// TIA Portal project "Connection" (V15.1)

(* hardware
DEVICE "S71500/ET200MP station_1"  S7-1500 station
   slot 0: "PM 190W 120/230VAC"  PM 190W 120/230VAC  6EP1333-4BA00
   slot 0: "Rail_0"  Rack  6ES7 590-1***0-0AA0
   slot 1: "PLC_1"  CPU 1516-3 PN/DP  6ES7 516-3AN01-0AB0  V2.6
      slot 3: "CPU display_1"  6ES7591-1BA00-0AA0
*)

// ===== PLC "PLC_1"  CPU 1516-3 PN/DP =====

VAR_GLOBAL   // PLC tag table "Default tag table"
   "System_Byte" AT %MB1 : Byte;
   "FirstScan" AT %M1.0 : Bool;
   "DiagStatusUpdate" AT %M1.1 : Bool;
   "AlwaysTRUE" AT %M1.2 : Bool;
   "AlwaysFALSE" AT %M1.3 : Bool;
   "Clock_Byte" AT %MB0 : Byte;
   "Clock_10Hz" AT %M0.0 : Bool;
   "Clock_5Hz" AT %M0.1 : Bool;
   "Clock_2.5Hz" AT %M0.2 : Bool;
   "Clock_2Hz" AT %M0.3 : Bool;
   "Clock_1.25Hz" AT %M0.4 : Bool;
   "Clock_1Hz" AT %M0.5 : Bool;
   "Clock_0.625Hz" AT %M0.6 : Bool;
   "Clock_0.5Hz" AT %M0.7 : Bool;
   "Connect" AT %M2.0 : Bool;
   "Reset" AT %M2.1 : Bool;
   "Send on/off" AT %M2.2 : Bool;
   "Receive enable" AT %M2.3 : Bool;
END_VAR

DATA_BLOCK "TCPIP_COMMS_DB"   // DB1
{ S7_Optimized_Access := 'TRUE' }
VERSION : 0.1
// stored: InstanceOfName TCPIP_COMMS
"TCPIP_COMMS"
BEGIN
END_DATA_BLOCK

DATA_BLOCK "Data"   // DB7
{ S7_Optimized_Access := 'TRUE' }
VERSION : 0.1
   VAR
      Recieving : Array[0..20] of Char;
      Sending : String := 'cc("Auto Position","AutoPositionAction","Pick And Place")\r\n';
   END_VAR
BEGIN
END_DATA_BLOCK

// folder: System blocks/Program resources

DATA_BLOCK "PLC_1_Connection_DB"   // DB3
{ S7_Optimized_Access := 'TRUE' }
AUTHOR : SIMATIC
FAMILY : MC7Plus
NAME : TC_IP_v4
VERSION : 1.0
// stored: InstanceOfName TCON_IP_v4
"TCON_IP_v4"
BEGIN
   ID := 1;
   InterfaceId := 64;
   LocalPort := 2000;
   RemotePort := 10999;
   ActiveEstablished := true;
   RemoteAddress.ADDR[1] := 192;
   RemoteAddress.ADDR[2] := 168;
   RemoteAddress.ADDR[4] := 3;
END_DATA_BLOCK

// folder: (top level)

FUNCTION_BLOCK "TCPIP_COMMS"   // FB1, LAD
{ S7_Optimized_Access := 'TRUE' }
VERSION : 0.1
   VAR
      TCON : Struct
         REQ : Bool;
         DONE : Bool;
         BUSY : Bool;
         ERROR : Bool;
         STATUS : UInt;
         DONESAVE : Bool;
         SAVED : Bool;
      END_STRUCT;
      TDISCON : Struct
         REQ : Bool;
         DONE : Bool;
         BUSY : Bool;
         ERROR : Bool;
         DONESAVE : Bool;
         STATUS : UInt;
      END_STRUCT;
      TSEND : Struct
         REQ : Bool;
         DONE : Bool;
         BUSY : Bool;
         ERROR : Bool;
         STATUS : UInt;
      END_STRUCT;
      TRCV : Struct
         EN_R : Bool;
         NDR : Bool;
         BUSY : Bool;
         ERROR : Bool;
         STATUS : UInt;
         RCVD_LEN : UDInt;
      END_STRUCT;
      "Received String" : String;
   END_VAR
BEGIN

REGION Network 1: TCON
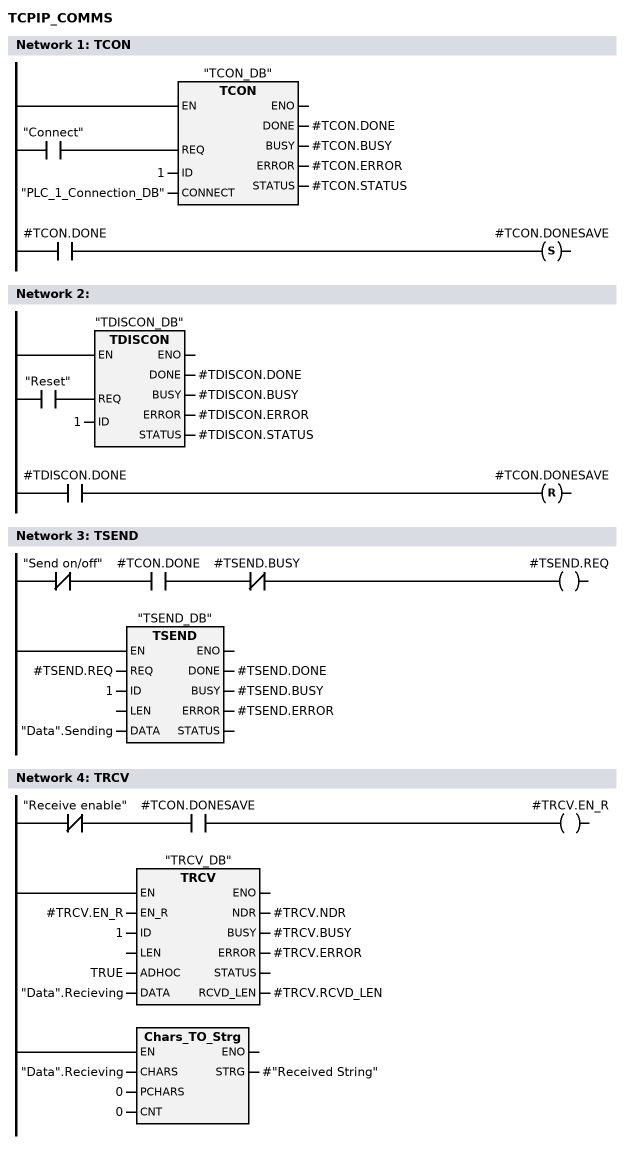
   "TCON_DB"(REQ := "Connect",   // TCON
             ID := 1,
             CONNECT := "PLC_1_Connection_DB",
             DONE => #TCON.DONE,
             BUSY => #TCON.BUSY,
             ERROR => #TCON.ERROR,
             STATUS => #TCON.STATUS);
   IF #TCON.DONE THEN #TCON.DONESAVE := TRUE; END_IF;
END_REGION

REGION Network 2
   "TDISCON_DB"(REQ := "Reset",   // TDISCON
                ID := 1,
                DONE => #TDISCON.DONE,
                BUSY => #TDISCON.BUSY,
                ERROR => #TDISCON.ERROR,
                STATUS => #TDISCON.STATUS);
   IF #TDISCON.DONE THEN #TCON.DONESAVE := FALSE; END_IF;
END_REGION

REGION Network 3: TSEND
   #TSEND.REQ := NOT "Send on/off" AND #TCON.DONE AND NOT #TSEND.BUSY;
   "TSEND_DB"(REQ := #TSEND.REQ,   // TSEND
              ID := 1,
              DATA := "Data".Sending,
              DONE => #TSEND.DONE,
              BUSY => #TSEND.BUSY,
              ERROR => #TSEND.ERROR);
END_REGION

REGION Network 4: TRCV
   // no SCL statement known for Chars_TO_Strg: written as a call
   #TRCV.EN_R := NOT "Receive enable" AND #TCON.DONESAVE;
   "TRCV_DB"(EN_R := #TRCV.EN_R,   // TRCV
             ID := 1,
             ADHOC := TRUE,
             DATA := "Data".Recieving,
             NDR => #TRCV.NDR,
             BUSY => #TRCV.BUSY,
             ERROR => #TRCV.ERROR,
             RCVD_LEN => #TRCV.RCVD_LEN);
   Chars_TO_Strg(Chars := "Data".Recieving, pChars := 0, Cnt := 0, Strg => #"Received String");
END_REGION
END_FUNCTION_BLOCK

ORGANIZATION_BLOCK "Main"   // OB1, LAD, ProgramCycle
TITLE = "Main Program Sweep (Cycle)"
{ S7_Optimized_Access := 'TRUE' }
VERSION : 0.1
   VAR_INPUT
      Initial_Call : Bool;   // Initial call of this OB
      Remanence : Bool;   // =True, if remanent data are available
   END_VAR
BEGIN

REGION Network 1
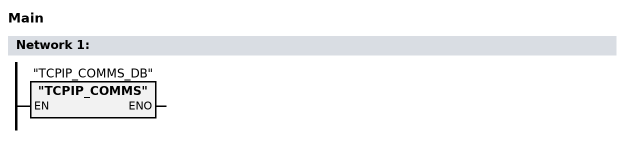
   RUNG wire#powerrail
      "TCPIP_COMMS_DB"()
   END_RUNG
   // the same network as SCL:
   "TCPIP_COMMS_DB"();   // "TCPIP_COMMS"
END_REGION
END_ORGANIZATION_BLOCK